(* Logix 5000 project; controller PBS_Perfusion vendor 1 type 14 code 217 rev 32.14; software revision 32.03; part 6 of 27 *)
(* tags used below, declared in another part *)
   Inp_PVSrcQ : DINT;   // Input Source and Quality (from Channel object, if available) (enum)
   Inp_PVNotify : DINT;   // Related PV object alarm prio and ack status (enum)
   Inp_PVBad : BOOL;   // 1=PV or I/O Comms Status Bad, 0=OK
   Inp_PVUncertain : BOOL;   // 1=PV Value Not Reliable, 0=OK
   Inp_Sim : BOOL;   // 1=Use simulated PV (Set_SimPV); 0=Use Input (Inp_PV)
   Cfg_HasRoC : BOOL;   // 1=Enables the Rate of Change calc and HiRoC alarm
   Cfg_HasDev : BOOL;   // 1=Enables Reference entry and Deviation calc and alarms
   Cfg_UseChanSrcQ : BOOL;   // 1=Pass thru connected Channel's SrcQ value, 0=generate SrcQ
   Cfg_RateTime : REAL;   // PV Rate of Change time base (sec) 60=/min, 3600=/hr
   Cfg_Ref : REAL;   // Analog Reference for Deviation Alarms (EU)
   Cfg_CtrlHiHiLim : REAL;   // Current High-High Control Threshold
   Cfg_CtrlHiHiDB : REAL;   // High-High Control Deadband (EU)
   Cfg_CtrlHiLim : REAL;   // Current High Control Threshold
   Cfg_CtrlHiDB : REAL;   // High Control Deadband (EU)
   Cfg_CtrlLoLim : REAL;   // Current Low Control Threshold
   Cfg_CtrlLoDB : REAL;   // Low Control Deadband (EU)
   Cfg_CtrlLoLoLim : REAL;   // Current Low-Low Control Threshold
   Cfg_CtrlLoLoDB : REAL;   // Low-Low Control Deadband (EU)
   Cfg_HiHiLim : REAL;   // Current High-High Status Threshold
   Cfg_HiHiDB : REAL;   // High-High Status Deadband (EU)
   Cfg_HiLim : REAL;   // Current High Status Threshold
   Cfg_HiDB : REAL;   // High Status Deadband (EU)
   Cfg_LoLim : REAL;   // Current Low Status Threshold
   Cfg_LoDB : REAL;   // Low Status Deadband (EU)
   Cfg_LoLoLim : REAL;   // Current Low-Low Status Threshold
   Cfg_LoLoDB : REAL;   // Low-Low Status Deadband (EU)
   Cfg_HiRoCLim : REAL;   // Current High Rate of Change Status Threshold
   Cfg_HiRoCDB : REAL;   // High Rate of Change Status Deadband (EU/rate time)
   Cfg_HiDevLim : REAL;   // Current High Deviation Status Threshold
   Cfg_HiDevDB : REAL;   // High Deviation Status Deadband (EU)
   Cfg_LoDevLim : REAL;   // Current Low Deviation Status Threshold
   Cfg_LoDevDB : REAL;   // Low Deviation Status Deadband (EU)
   Cfg_FailHiLim : REAL;   // Out-of-Range (fail) High Limit (EU)
   Cfg_FailLoLim : REAL;   // Out-of-Range (fail) Low Limit (EU)
   Cfg_FailDB : REAL;   // Out-of-Range (fail) High/Low Deadband (EU)
   PCmd_ClearCapt : BOOL;   // Program Command to Clear the captured min / max PV excursion values
   Val : REAL;   // Analog Input Value (incl. Manual Override, if used)
   Val_InpPV : REAL;   // Analog Input Value (actual, before Substitute PV selection)
   Val_RoC : REAL;   // Analog Value Rate of Change (EU/rate time)
   Val_Dev : REAL;   // Calculated Deviation from Reference (EU)
   Val_PVMinCapt : REAL;   // Captured PV Minimum (excursion) since last cleared
   Val_PVMaxCapt : REAL;   // Captured PV Maximum (excursion) since last cleared
   SrcQ_IO : DINT;   // Source and Quality of primary I/O (enumeration)
   SrcQ : DINT;   // Source and Quality of primary Val/Sts (enumeration)
   Val_Fault : DINT;   // Device Fault Status 0=none, 20=Lo, 21=Hi, 22=LoDev, 23=HiDev, 24=LoLo, 25=HiHi, 26=HiRoC 32=Fail, 34=CfgErr
   Val_NotifyAll : DINT;   // Highest Alarm prio and ack status this object + channel (enum)
   Val_UnackAlmC : DINT;   // Count of Unacknowledged Alarms
   Sts_SubstPV : BOOL;   // 1=Using Substitute PV (Input being overridden)
   Sts_PVBad : BOOL;   // 1=PV Bad quality or Out of Range
   Sts_PVUncertain : BOOL;   // 1=PV Value is Uncertain (quality)
   Sts_AlmInh : BOOL;   // 1=An Alarm is Shelved, Disabled or Suppressed: display icon
   Sts_Err : BOOL;   // 1=Error in Config: see detail bits for reason
   Err_Raw : BOOL;   // 1=Error in Config: Raw Input Scaling Min = Max
   Err_EU : BOOL;   // 1=Error in Config: Scaled EU Min = Max
   Err_Timer : BOOL;   // 1=Error in Config: On-Delay, Off-Delay, Gate Delay Time Invalid (use 0 to 2147483 s)
   Err_Filt : BOOL;   // 1=-Error in Config: PV filter params (RateTime, TC)
   Err_Alarm : BOOL;   // 1=Error in Config: Alarm Min On Time, Shelf Time, Severity
   Sts_RdyReset : ALIAS FOR ORdy_Reset;   // 1=A latched alarm or shed condition is ready to be reset
   Sts_RdyAck : BOOL;   // 1=An alarm is ready to be acknowledged
   Sts_CtrlHiHi : BOOL;   // 1=Analog Input is above High-High Control limit
   Sts_CtrlHi : BOOL;   // 1=Analog Input is above High Control limit
   Sts_CtrlLo : BOOL;   // 1=Analog Input is above Low Control limit
   Sts_CtrlLoLo : BOOL;   // 1=Analog Input is above Low-Low Control limit
   Sts_HiHiCmp : ALIAS FOR HiHiGate.Inp;   // PV High-High comparison result 1=High-High
   Sts_HiHi : ALIAS FOR HiHi.Inp;   // 1=Analog Input is above High-High limit
   Sts_HiCmp : ALIAS FOR HiGate.Inp;   // PV High comparison result 1=High
   Sts_Hi : ALIAS FOR Hi.Inp;   // 1=Analog Input is above High limit
   Sts_LoCmp : ALIAS FOR LoGate.Inp;   // PV Low comparison result 1=Low
   Sts_Lo : ALIAS FOR Lo.Inp;   // 1=Analog Input is below Low limit
   Sts_LoLoCmp : ALIAS FOR LoLoGate.Inp;   // PV Low-Low comparison result 1=Low-Low
   Sts_LoLo : ALIAS FOR LoLo.Inp;   // 1=Analog Input is below Low-Low limit
   Sts_HiRoCCmp : ALIAS FOR HiRoCGate.Inp;   // PV High Rate of Change comparison result 1=High
   Sts_HiRoC : ALIAS FOR HiRoC.Inp;   // 1=Analog Input Rate of Change is above High limit
   Sts_HiDevCmp : ALIAS FOR HiDevGate.Inp;   // PV High Deviation comparison result 1=Dev High
   Sts_HiDev : ALIAS FOR HiDev.Inp;   // 1=Analog Input Deviation is above High limit
   Sts_LoDevCmp : ALIAS FOR LoDevGate.Inp;   // PV Low Deviation comparison result 1=Dev Low
   Sts_LoDev : ALIAS FOR LoDev.Inp;   // 1=Analog Input Deviation is below Low limit
   Sts_FailCmp : ALIAS FOR FailGate.Inp;   // PV Fail comparison result 1=Out of Range
   Sts_Fail : ALIAS FOR Fail.Inp;   // 1=Analog Input is Out of Range or PV Bad
   P_AInAdv : BOOL;   // Unique Parameter Name for auto - discovery
   LoLo : P_Alarm;   // Low-Low Alarm
   Lo : P_Alarm;   // Low Alarm
   Hi : P_Alarm;   // High Alarm
   HiHi : P_Alarm;   // High-High Alarm
   Fail : P_Alarm;   // Analog Input Failure Alarm (bad quality or out of range)
   Wrk_Notify : DINT;   // Buffer for building Val_Notify
   Wrk_Fault : DINT;   // Buffer for building Val_Fault
   Wrk_SrcQ : DINT;   // Register for building Source / Quality enumeration
   Wrk_SubstPV : BOOL;   // Internal flag: Using Substitute PV
   Wrk_ScanTime : REAL;   // Time since this instance was last scanned
   Wrk_RoC : REAL;   // Calculated Rate of Change of PV
   Wrk_PrevPV : REAL;   // Previous scan's value of Filtered PV
   LoDev : P_Alarm;   // Low Deviation Alarm
   HiDev : P_Alarm;   // High Deviation Alarm
   HiRoC : P_Alarm;   // High Rate of Change Alarm
   Wrk_InpInfNaN : BOOL;   // Input (Inp_PV or Set_SimPV) Infinite or Not a Number
   Wrk_SelPVInfNaN : BOOL;   // Selected PV (Input or Substitute) is Infinite or NaN
   Wrk_HiRoC : BOOL;   // Internal flag: High Rate of Change Status
   Wrk_LoDev : BOOL;   // Internal flag: Low Deviation Status
   Wrk_HiDev : BOOL;   // Internal flag: High Deviation Status
   Wrk_Fail : BOOL;   // Internal flag: Fail Status
   Wrk_LoLo : BOOL;   // Internal flag: Low-Low Status
   Wrk_Lo : BOOL;   // Internal flag: Low Status
   Wrk_HiHi : BOOL;   // Internal flag: High-High Status
   Wrk_Hi : BOOL;   // Internal flag: High Status
   LoDevGate : P_Gate;   // Low Deviation Alarm Gate / Delay Block
   HiRoCGate : P_Gate;   // High Rate of Change Alarm Gate / Delay Block
   HiDevGate : P_Gate;   // High Deviation Alarm Gate / Delay Block
   LoLoGate : P_Gate;   // Low-Low Alarm Gate / Delay Block
   LoGate : P_Gate;   // Low Alarm Gate / Delay Block
   HiHiGate : P_Gate;   // High-High Alarm Gate / Delay Block
   HiGate : P_Gate;   // High Alarm Gate / Delay Block
   FailGate : P_Gate;   // Fail Alarm Gate / Delay Block
   Wrk_UnackAlmC : DINT;   // Buffer for building Val_UnackAlmC
   Val_Notify : DINT;   // Highest Alarm prio and ack status this object only (enum)
   OCmd_ClearCapt : BOOL;   // Operator Command to Clear the captured min / max PV excursion values
   ORdy_ResetAckAll : BOOL;   // 1=Ready for OCmd_ResetAckAll (enables HMI button)
   ORdy_Reset : BOOL;   // 1=Ready for OCmd_Reset (enables HMI button)
   Wrk_RawPV : REAL;   // Value of raw PV to be used for Out of Range checking
   REAL : DINT;
(* P_AInAdv, continued *)

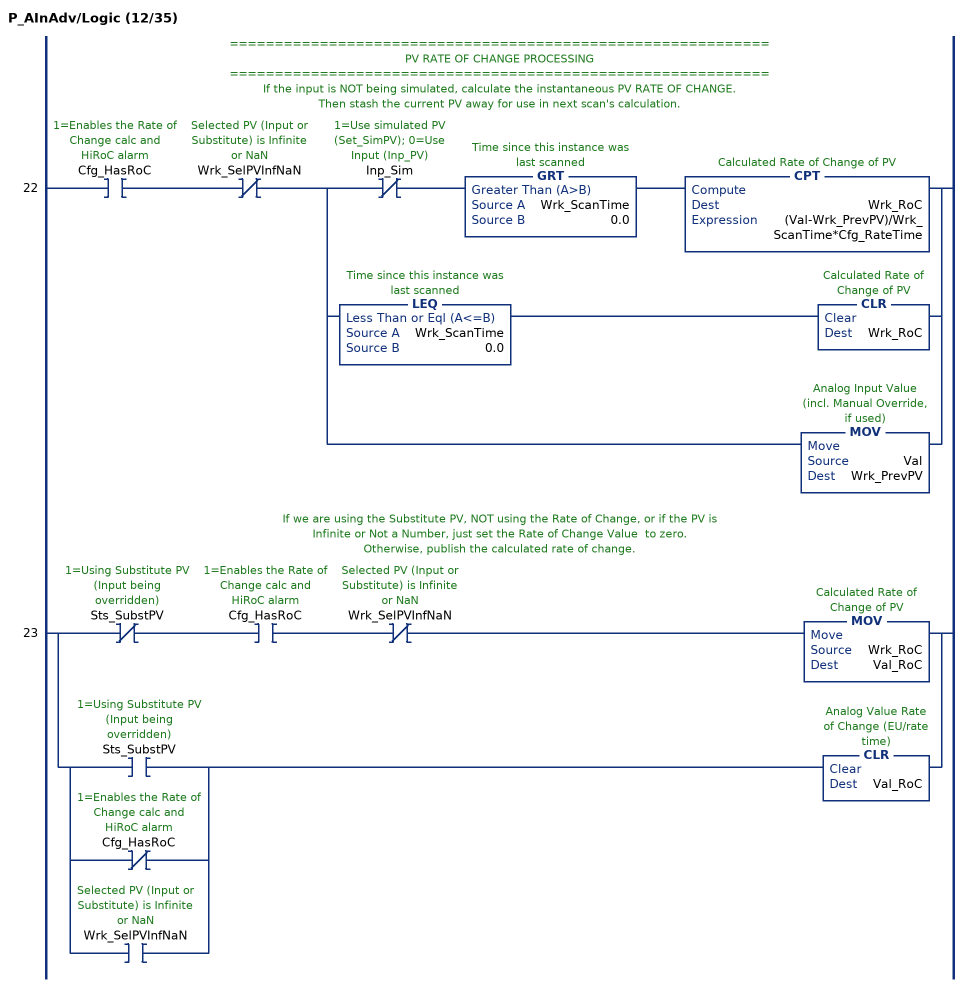
   [picture p107: P_AInAdv/Logic rungs 22-23]
   // ============================================================
   // PV RATE OF CHANGE PROCESSING
   // ============================================================
   // If the input is NOT being simulated, calculate the instantaneous PV RATE OF CHANGE.
   // Then stash the current PV away for use in next scan's calculation.
   22: XIC(Cfg_HasRoC)XIO(Wrk_SelPVInfNaN)[XIO(Inp_Sim) GRT(Wrk_ScanTime,0.0) CPT(Wrk_RoC,(Val-Wrk_PrevPV)/Wrk_ScanTime*Cfg_RateTime) ,LEQ(Wrk_ScanTime,0.0) CLR(Wrk_RoC) ,MOV(Val,Wrk_PrevPV) ];
   // If we are using the Substitute PV, NOT using the Rate of Change, or if the PV is
   // Infinite or Not a Number, just set the Rate of Change Value  to zero.
   // Otherwise, publish the calculated rate of change.
   23: [XIO(Sts_SubstPV) XIC(Cfg_HasRoC) XIO(Wrk_SelPVInfNaN) MOV(Wrk_RoC,Val_RoC) ,[XIC(Sts_SubstPV) ,XIO(Cfg_HasRoC) ,XIC(Wrk_SelPVInfNaN) ] CLR(Val_RoC) ];
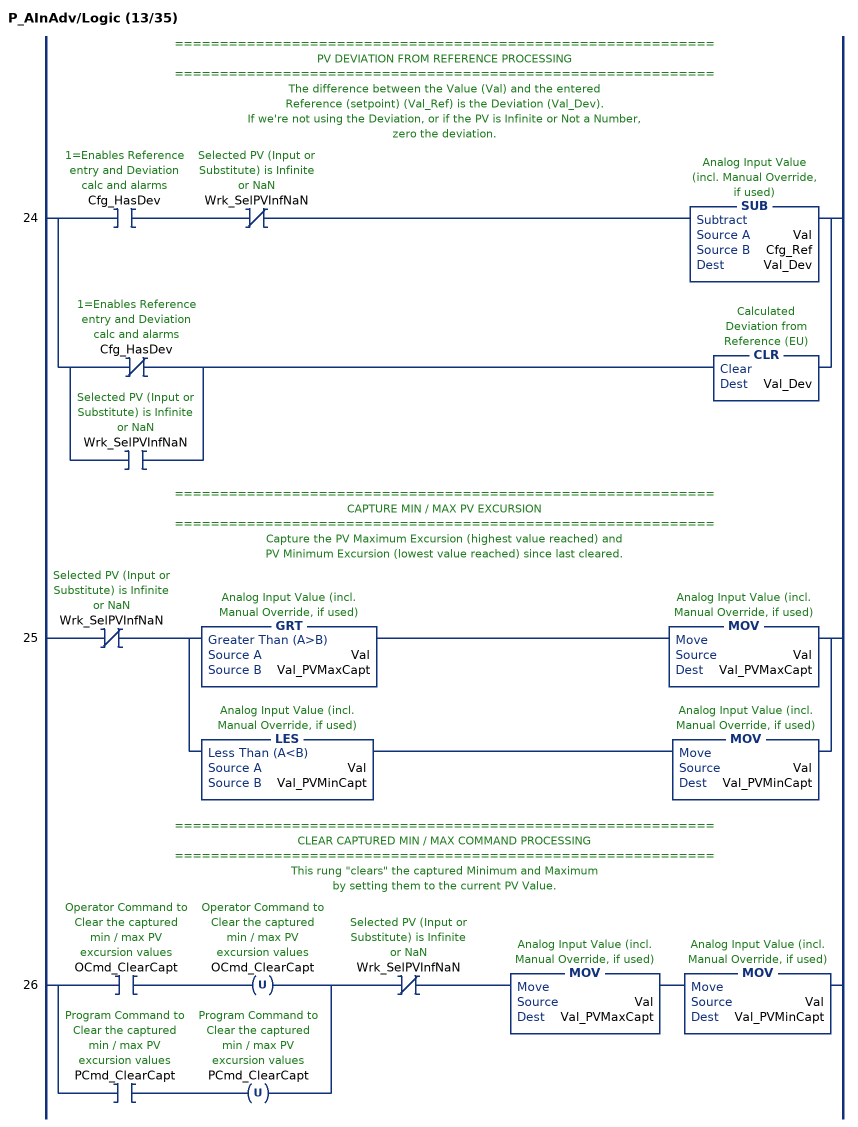
   // ============================================================
   // PV DEVIATION FROM REFERENCE PROCESSING
   // ============================================================
   // The difference between the Value (Val) and the entered
   // Reference (setpoint) (Val_Ref) is the Deviation (Val_Dev).
   // If we're not using the Deviation, or if the PV is Infinite or Not a Number,
   // zero the deviation.
   24: [XIC(Cfg_HasDev) XIO(Wrk_SelPVInfNaN) SUB(Val,Cfg_Ref,Val_Dev) ,[XIO(Cfg_HasDev) ,XIC(Wrk_SelPVInfNaN) ] CLR(Val_Dev) ];
   // ============================================================
   // CAPTURE MIN / MAX PV EXCURSION
   // ============================================================
   // Capture the PV Maximum Excursion (highest value reached) and
   // PV Minimum Excursion (lowest value reached) since last cleared.
   25: XIO(Wrk_SelPVInfNaN)[GRT(Val,Val_PVMaxCapt) MOV(Val,Val_PVMaxCapt) ,LES(Val,Val_PVMinCapt) MOV(Val,Val_PVMinCapt) ];
   // ============================================================
   // CLEAR CAPTURED MIN / MAX COMMAND PROCESSING
   // ============================================================
   // This rung "clears" the captured Minimum and Maximum
   // by setting them to the current PV Value.
   26: [XIC(OCmd_ClearCapt) OTU(OCmd_ClearCapt) ,XIC(PCmd_ClearCapt) OTU(PCmd_ClearCapt) ]XIO(Wrk_SelPVInfNaN)MOV(Val,Val_PVMaxCapt)MOV(Val,Val_PVMinCapt);
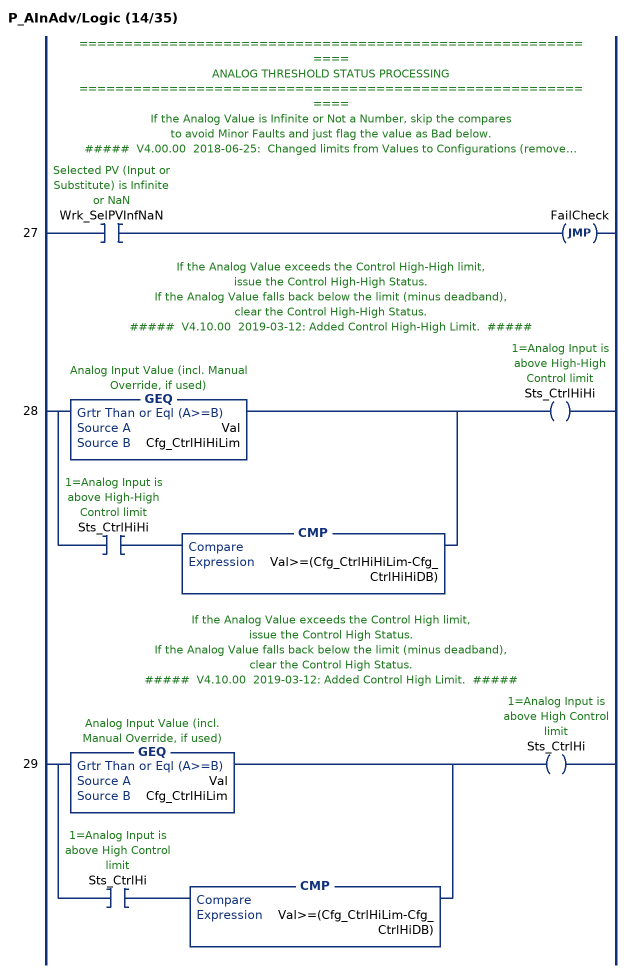
   // ============================================================
   // ANALOG THRESHOLD STATUS PROCESSING
   // ============================================================
   // If the Analog Value is Infinite or Not a Number, skip the compares
   // to avoid Minor Faults and just flag the value as Bad below.
   // #####  V4.00.00  2018-06-25:  Changed limits from Values to Configurations (removed Mode, Settings).  #####
   // #####  Changed PV Out of Range comparisons to use RAW (INPUT) PV, not scaled/filtered value (Val).  #####
   27: XIC(Wrk_SelPVInfNaN)JMP(FailCheck);
   // If the Analog Value exceeds the Control High-High limit,
   // issue the Control High-High Status.
   // If the Analog Value falls back below the limit (minus deadband),
   // clear the Control High-High Status.
   // #####  V4.10.00  2019-03-12: Added Control High-High Limit.  #####
   28: [GEQ(Val,Cfg_CtrlHiHiLim) ,XIC(Sts_CtrlHiHi) CMP(Val>=(Cfg_CtrlHiHiLim-Cfg_CtrlHiHiDB)) ]OTE(Sts_CtrlHiHi);
   // If the Analog Value exceeds the Control High limit,
   // issue the Control High Status.
   // If the Analog Value falls back below the limit (minus deadband),
   // clear the Control High Status.
   // #####  V4.10.00  2019-03-12: Added Control High Limit.  #####
   29: [GEQ(Val,Cfg_CtrlHiLim) ,XIC(Sts_CtrlHi) CMP(Val>=(Cfg_CtrlHiLim-Cfg_CtrlHiDB)) ]OTE(Sts_CtrlHi);
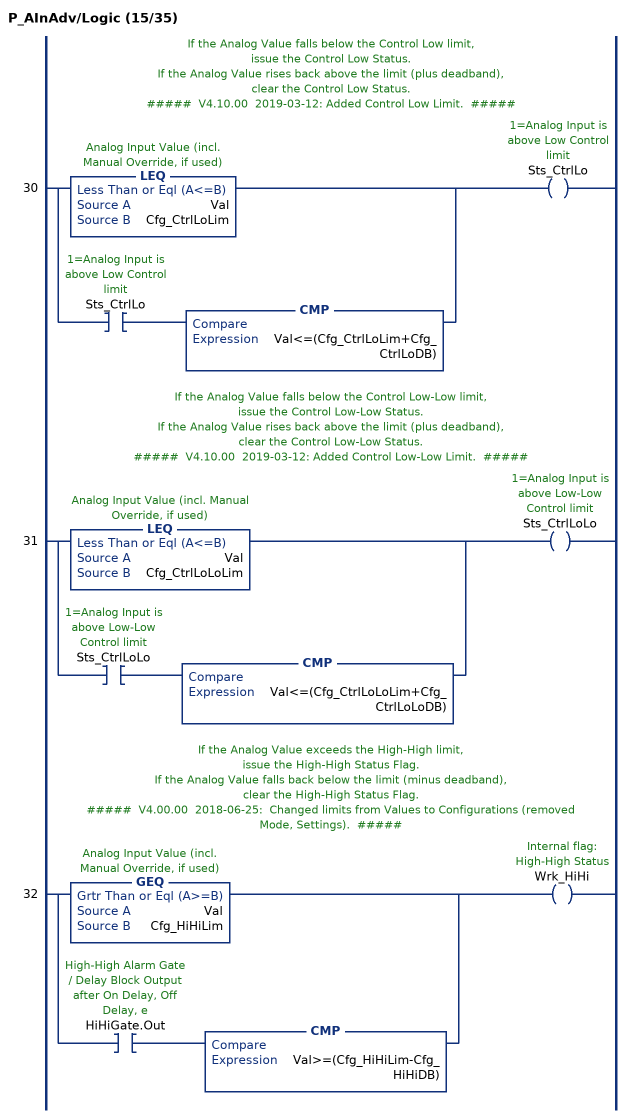
   // If the Analog Value falls below the Control Low limit,
   // issue the Control Low Status.
   // If the Analog Value rises back above the limit (plus deadband),
   // clear the Control Low Status.
   // #####  V4.10.00  2019-03-12: Added Control Low Limit.  #####
   30: [LEQ(Val,Cfg_CtrlLoLim) ,XIC(Sts_CtrlLo) CMP(Val<=(Cfg_CtrlLoLim+Cfg_CtrlLoDB)) ]OTE(Sts_CtrlLo);
   // If the Analog Value falls below the Control Low-Low limit,
   // issue the Control Low-Low Status.
   // If the Analog Value rises back above the limit (plus deadband),
   // clear the Control Low-Low Status.
   // #####  V4.10.00  2019-03-12: Added Control Low-Low Limit.  #####
   31: [LEQ(Val,Cfg_CtrlLoLoLim) ,XIC(Sts_CtrlLoLo) CMP(Val<=(Cfg_CtrlLoLoLim+Cfg_CtrlLoLoDB)) ]OTE(Sts_CtrlLoLo);
   // If the Analog Value exceeds the High-High limit,
   // issue the High-High Status Flag.
   // If the Analog Value falls back below the limit (minus deadband),
   // clear the High-High Status Flag.
   // #####  V4.00.00  2018-06-25:  Changed limits from Values to Configurations (removed Mode, Settings).  #####
   32: [GEQ(Val,Cfg_HiHiLim) ,XIC(HiHiGate.Out) CMP(Val>=(Cfg_HiHiLim-Cfg_HiHiDB)) ]OTE(Wrk_HiHi);
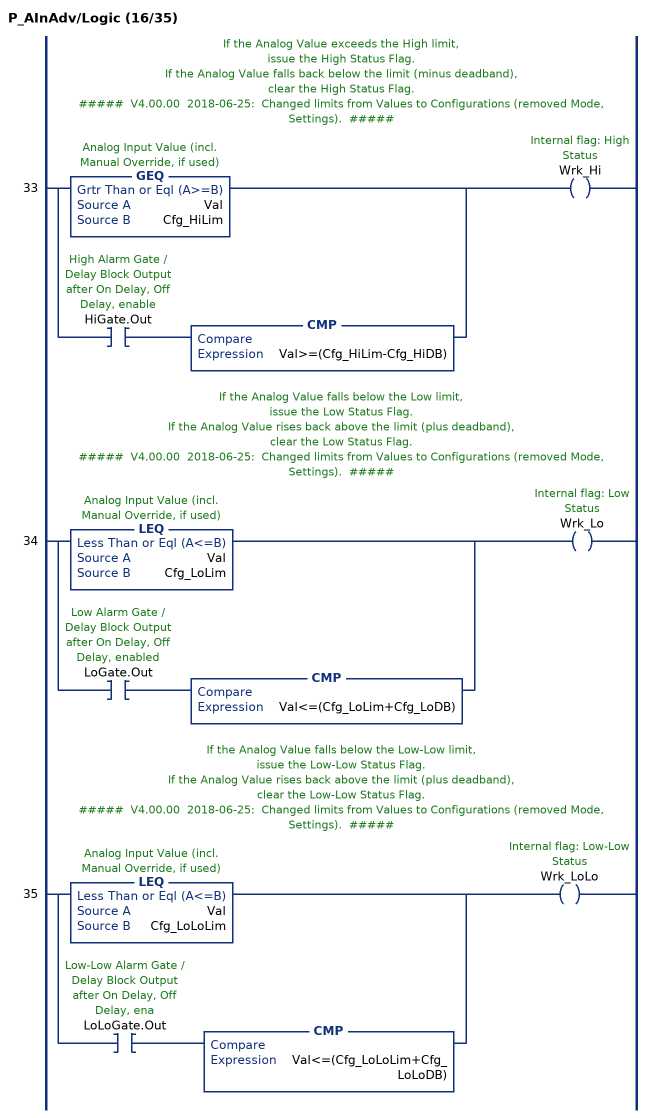
   // If the Analog Value exceeds the High limit,
   // issue the High Status Flag.
   // If the Analog Value falls back below the limit (minus deadband),
   // clear the High Status Flag.
   // #####  V4.00.00  2018-06-25:  Changed limits from Values to Configurations (removed Mode, Settings).  #####
   33: [GEQ(Val,Cfg_HiLim) ,XIC(HiGate.Out) CMP(Val>=(Cfg_HiLim-Cfg_HiDB)) ]OTE(Wrk_Hi);
   // If the Analog Value falls below the Low limit,
   // issue the Low Status Flag.
   // If the Analog Value rises back above the limit (plus deadband),
   // clear the Low Status Flag.
   // #####  V4.00.00  2018-06-25:  Changed limits from Values to Configurations (removed Mode, Settings).  #####
   34: [LEQ(Val,Cfg_LoLim) ,XIC(LoGate.Out) CMP(Val<=(Cfg_LoLim+Cfg_LoDB)) ]OTE(Wrk_Lo);
   // If the Analog Value falls below the Low-Low limit,
   // issue the Low-Low Status Flag.
   // If the Analog Value rises back above the limit (plus deadband),
   // clear the Low-Low Status Flag.
   // #####  V4.00.00  2018-06-25:  Changed limits from Values to Configurations (removed Mode, Settings).  #####
   35: [LEQ(Val,Cfg_LoLoLim) ,XIC(LoLoGate.Out) CMP(Val<=(Cfg_LoLoLim+Cfg_LoLoDB)) ]OTE(Wrk_LoLo);
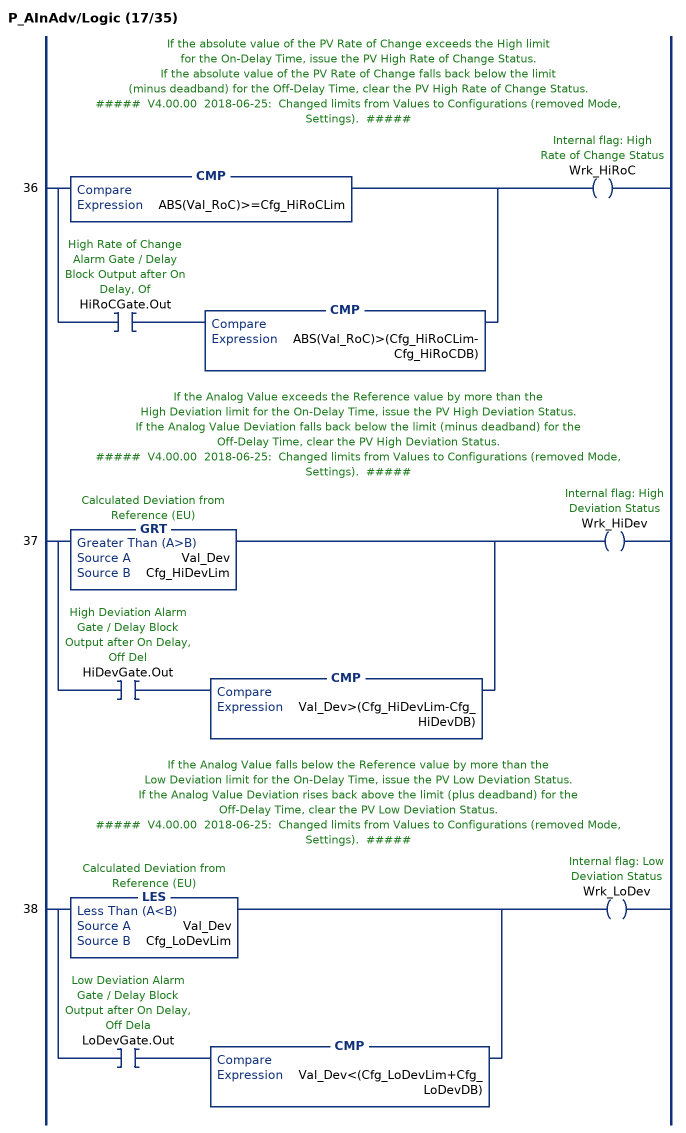
   // If the absolute value of the PV Rate of Change exceeds the High limit
   // for the On-Delay Time, issue the PV High Rate of Change Status.
   // If the absolute value of the PV Rate of Change falls back below the limit
   // (minus deadband) for the Off-Delay Time, clear the PV High Rate of Change Status.
   // #####  V4.00.00  2018-06-25:  Changed limits from Values to Configurations (removed Mode, Settings).  #####
   36: [CMP(ABS(Val_RoC)>=Cfg_HiRoCLim) ,XIC(HiRoCGate.Out) CMP(ABS(Val_RoC)>(Cfg_HiRoCLim-Cfg_HiRoCDB)) ]OTE(Wrk_HiRoC);
   // If the Analog Value exceeds the Reference value by more than the
   // High Deviation limit for the On-Delay Time, issue the PV High Deviation Status.
   // If the Analog Value Deviation falls back below the limit (minus deadband) for the
   // Off-Delay Time, clear the PV High Deviation Status.
   // #####  V4.00.00  2018-06-25:  Changed limits from Values to Configurations (removed Mode, Settings).  #####
   37: [GRT(Val_Dev,Cfg_HiDevLim) ,XIC(HiDevGate.Out) CMP(Val_Dev>(Cfg_HiDevLim-Cfg_HiDevDB)) ]OTE(Wrk_HiDev);
   // If the Analog Value falls below the Reference value by more than the
   // Low Deviation limit for the On-Delay Time, issue the PV Low Deviation Status.
   // If the Analog Value Deviation rises back above the limit (plus deadband) for the
   // Off-Delay Time, clear the PV Low Deviation Status.
   // #####  V4.00.00  2018-06-25:  Changed limits from Values to Configurations (removed Mode, Settings).  #####
   38: [LES(Val_Dev,Cfg_LoDevLim) ,XIC(LoDevGate.Out) CMP(Val_Dev<(Cfg_LoDevLim+Cfg_LoDevDB)) ]OTE(Wrk_LoDev);
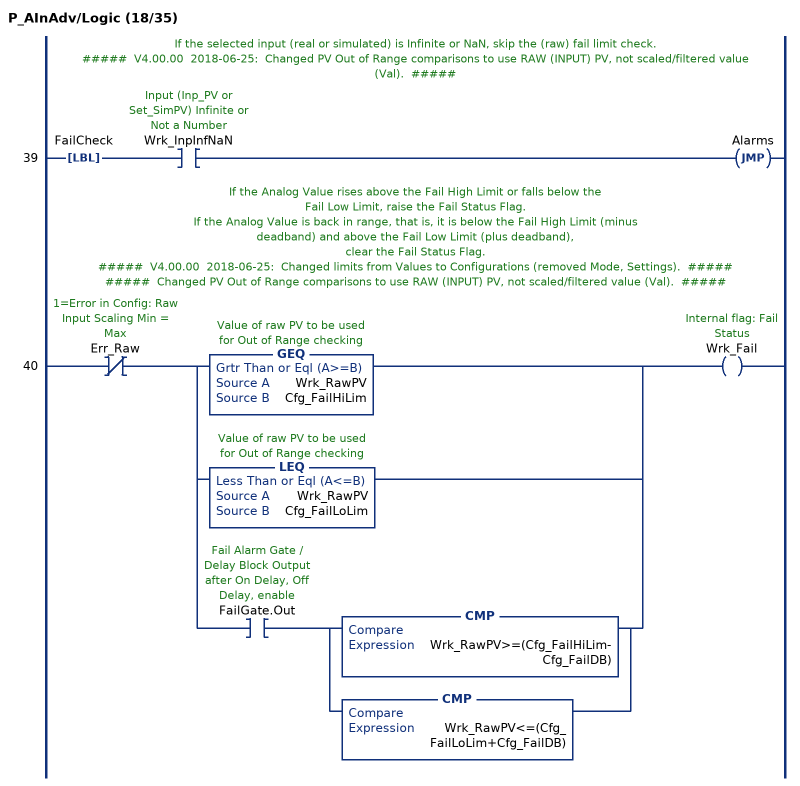
   // If the selected input (real or simulated) is Infinite or NaN, skip the (raw) fail limit check.
   // #####  V4.00.00  2018-06-25:  Changed PV Out of Range comparisons to use RAW (INPUT) PV, not scaled/filtered value (Val).  #####
   39: LBL(FailCheck)XIC(Wrk_InpInfNaN)JMP(Alarms);
   // If the Analog Value rises above the Fail High Limit or falls below the
   // Fail Low Limit, raise the Fail Status Flag.
   // If the Analog Value is back in range, that is, it is below the Fail High Limit (minus
   // deadband) and above the Fail Low Limit (plus deadband),
   // clear the Fail Status Flag.
   // #####  V4.00.00  2018-06-25:  Changed limits from Values to Configurations (removed Mode, Settings).  #####
   // #####  Changed PV Out of Range comparisons to use RAW (INPUT) PV, not scaled/filtered value (Val).  #####
   40: XIO(Err_Raw)[[GEQ(Wrk_RawPV,Cfg_FailHiLim) ,LEQ(Wrk_RawPV,Cfg_FailLoLim) ] ,XIC(FailGate.Out) [CMP(Wrk_RawPV>=(Cfg_FailHiLim-Cfg_FailDB)) ,CMP(Wrk_RawPV<=(Cfg_FailLoLim+Cfg_FailDB)) ] ]OTE(Wrk_Fail);
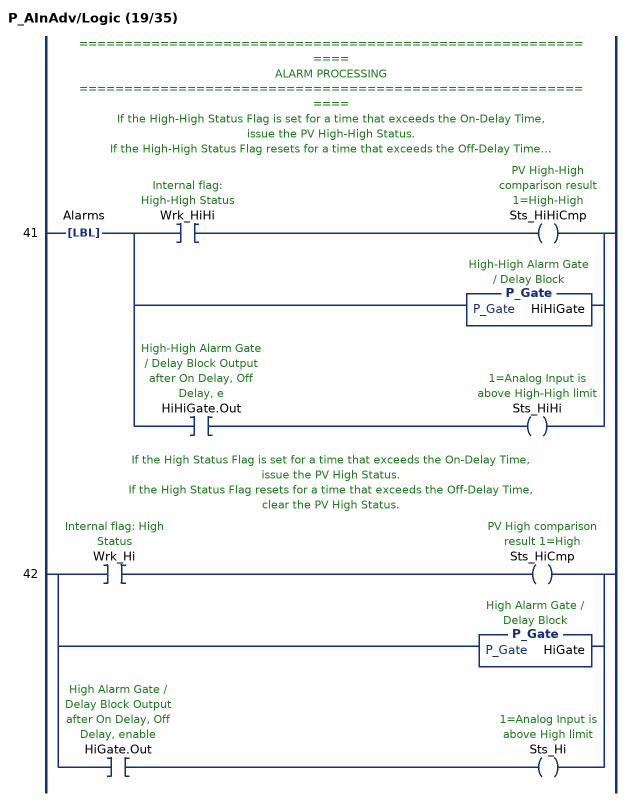
   // ============================================================
   // ALARM PROCESSING
   // ============================================================
   // If the High-High Status Flag is set for a time that exceeds the On-Delay Time,
   // issue the PV High-High Status.
   // If the High-High Status Flag resets for a time that exceeds the Off-Delay Time,
   // clear the PV High-High Status.
   41: LBL(Alarms)[XIC(Wrk_HiHi) OTE(Sts_HiHiCmp) ,P_Gate(HiHiGate) ,XIC(HiHiGate.Out) OTE(Sts_HiHi) ];
   // If the High Status Flag is set for a time that exceeds the On-Delay Time,
   // issue the PV High Status.
   // If the High Status Flag resets for a time that exceeds the Off-Delay Time,
   // clear the PV High Status.
   42: [XIC(Wrk_Hi) OTE(Sts_HiCmp) ,P_Gate(HiGate) ,XIC(HiGate.Out) OTE(Sts_Hi) ];
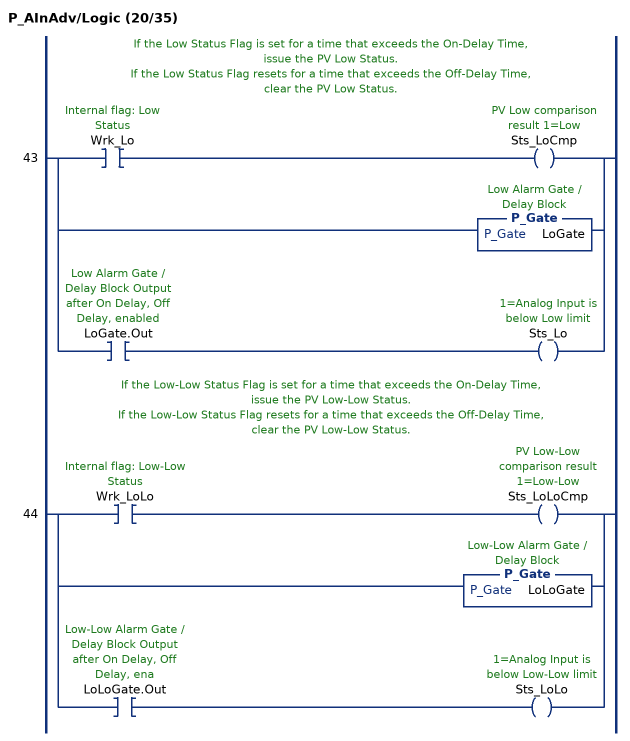
   // If the Low Status Flag is set for a time that exceeds the On-Delay Time,
   // issue the PV Low Status.
   // If the Low Status Flag resets for a time that exceeds the Off-Delay Time,
   // clear the PV Low Status.
   43: [XIC(Wrk_Lo) OTE(Sts_LoCmp) ,P_Gate(LoGate) ,XIC(LoGate.Out) OTE(Sts_Lo) ];
   // If the Low-Low Status Flag is set for a time that exceeds the On-Delay Time,
   // issue the PV Low-Low Status.
   // If the Low-Low Status Flag resets for a time that exceeds the Off-Delay Time,
   // clear the PV Low-Low Status.
   44: [XIC(Wrk_LoLo) OTE(Sts_LoLoCmp) ,P_Gate(LoLoGate) ,XIC(LoLoGate.Out) OTE(Sts_LoLo) ];
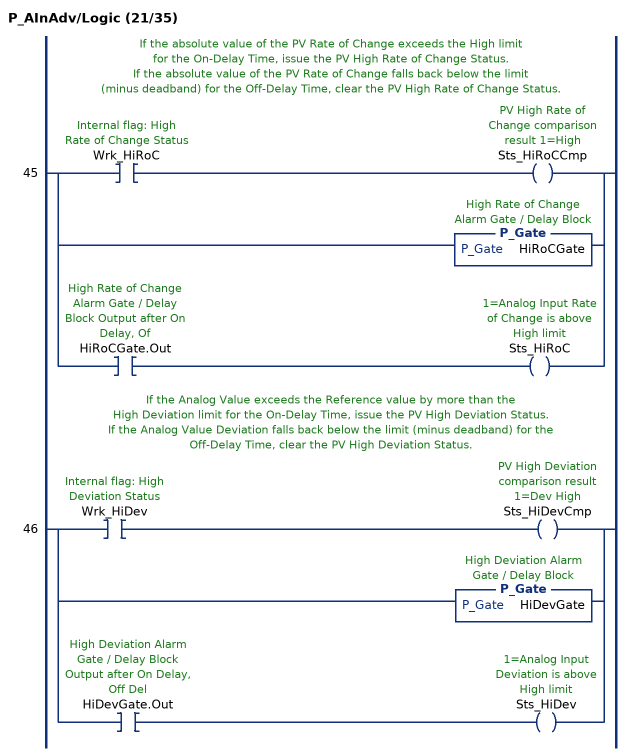
   // If the absolute value of the PV Rate of Change exceeds the High limit
   // for the On-Delay Time, issue the PV High Rate of Change Status.
   // If the absolute value of the PV Rate of Change falls back below the limit
   // (minus deadband) for the Off-Delay Time, clear the PV High Rate of Change Status.
   45: [XIC(Wrk_HiRoC) OTE(Sts_HiRoCCmp) ,P_Gate(HiRoCGate) ,XIC(HiRoCGate.Out) OTE(Sts_HiRoC) ];
   // If the Analog Value exceeds the Reference value by more than the
   // High Deviation limit for the On-Delay Time, issue the PV High Deviation Status.
   // If the Analog Value Deviation falls back below the limit (minus deadband) for the
   // Off-Delay Time, clear the PV High Deviation Status.
   46: [XIC(Wrk_HiDev) OTE(Sts_HiDevCmp) ,P_Gate(HiDevGate) ,XIC(HiDevGate.Out) OTE(Sts_HiDev) ];
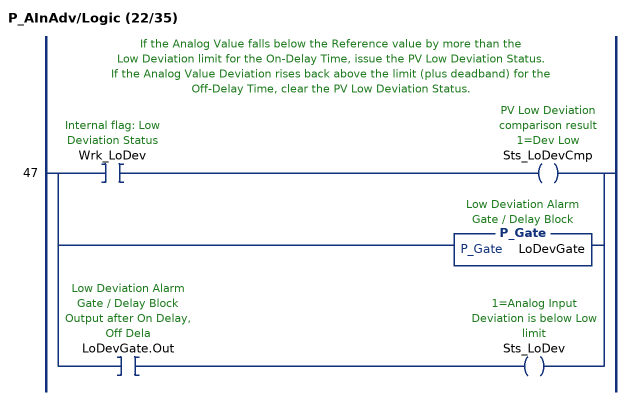
   // If the Analog Value falls below the Reference value by more than the
   // Low Deviation limit for the On-Delay Time, issue the PV Low Deviation Status.
   // If the Analog Value Deviation rises back above the limit (plus deadband) for the
   // Off-Delay Time, clear the PV Low Deviation Status.
   47: [XIC(Wrk_LoDev) OTE(Sts_LoDevCmp) ,P_Gate(LoDevGate) ,XIC(LoDevGate.Out) OTE(Sts_LoDev) ];
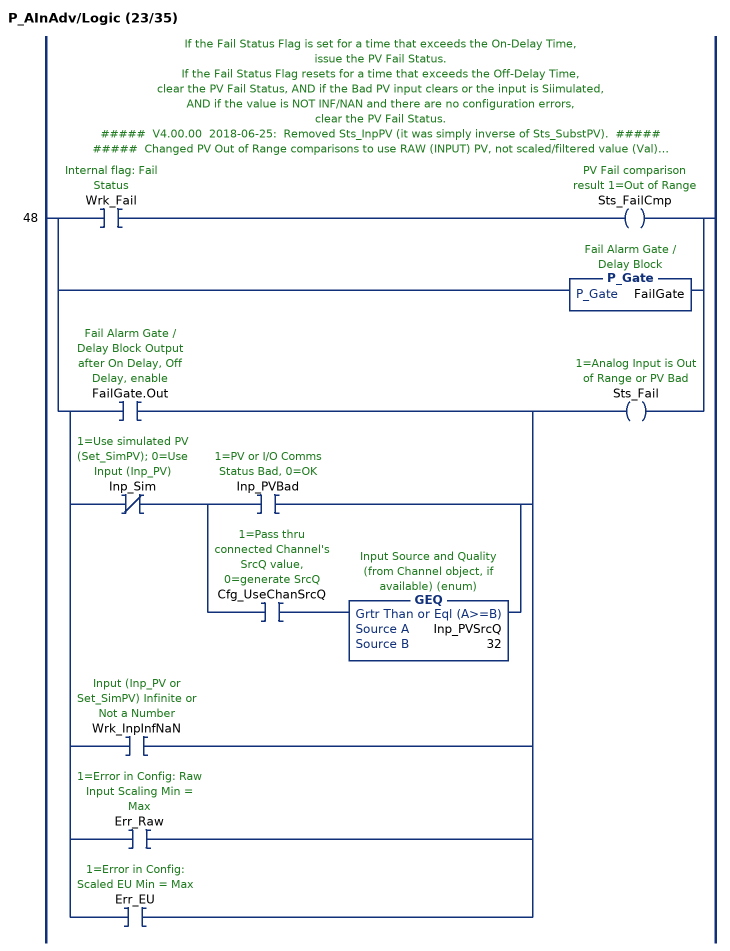
   // If the Fail Status Flag is set for a time that exceeds the On-Delay Time,
   // issue the PV Fail Status.
   // If the Fail Status Flag resets for a time that exceeds the Off-Delay Time,
   // clear the PV Fail Status, AND if the Bad PV input clears or the input is Siimulated,
   // AND if the value is NOT INF/NAN and there are no configuration errors,
   // clear the PV Fail Status.
   // #####  V4.00.00  2018-06-25:  Removed Sts_InpPV (it was simply inverse of Sts_SubstPV).  #####
   // #####  Changed PV Out of Range comparisons to use RAW (INPUT) PV, not scaled/filtered value (Val).  #####
   48: [XIC(Wrk_Fail) OTE(Sts_FailCmp) ,P_Gate(FailGate) ,[XIC(FailGate.Out) ,XIO(Inp_Sim) [XIC(Inp_PVBad) ,XIC(Cfg_UseChanSrcQ) GEQ(Inp_PVSrcQ,32) ] ,XIC(Wrk_InpInfNaN) ,XIC(Err_Raw) ,XIC(Err_EU) ] OTE(Sts_Fail) ];
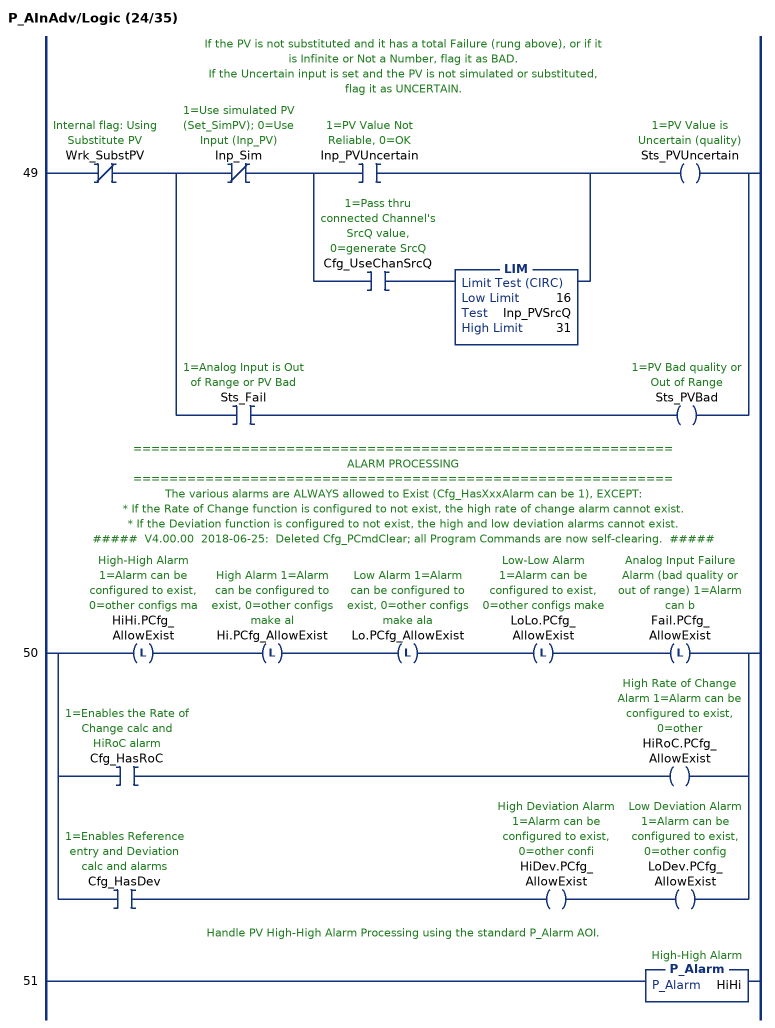
   // If the PV is not substituted and it has a total Failure (rung above), or if it
   // is Infinite or Not a Number, flag it as BAD.
   // If the Uncertain input is set and the PV is not simulated or substituted,
   // flag it as UNCERTAIN.
   49: XIO(Wrk_SubstPV)[XIO(Inp_Sim) [XIC(Inp_PVUncertain) ,XIC(Cfg_UseChanSrcQ) LIM(16,Inp_PVSrcQ,31) ] OTE(Sts_PVUncertain) ,XIC(Sts_Fail) OTE(Sts_PVBad) ];
   // ============================================================
   // ALARM PROCESSING
   // ============================================================
   // The various alarms are ALWAYS allowed to Exist (Cfg_HasXxxAlarm can be 1), EXCEPT:
   // * If the Rate of Change function is configured to not exist, the high rate of change alarm cannot exist.
   // * If the Deviation function is configured to not exist, the high and low deviation alarms cannot exist.
   // #####  V4.00.00  2018-06-25:  Deleted Cfg_PCmdClear; all Program Commands are now self-clearing.  #####
   50: [OTL(HiHi.PCfg_AllowExist) OTL(Hi.PCfg_AllowExist) OTL(Lo.PCfg_AllowExist) OTL(LoLo.PCfg_AllowExist) OTL(Fail.PCfg_AllowExist) ,XIC(Cfg_HasRoC) OTE(HiRoC.PCfg_AllowExist) ,XIC(Cfg_HasDev) OTE(HiDev.PCfg_AllowExist) OTE(LoDev.PCfg_AllowExist) ];
   // Handle PV High-High Alarm Processing using the standard P_Alarm AOI.
   51: P_Alarm(HiHi);
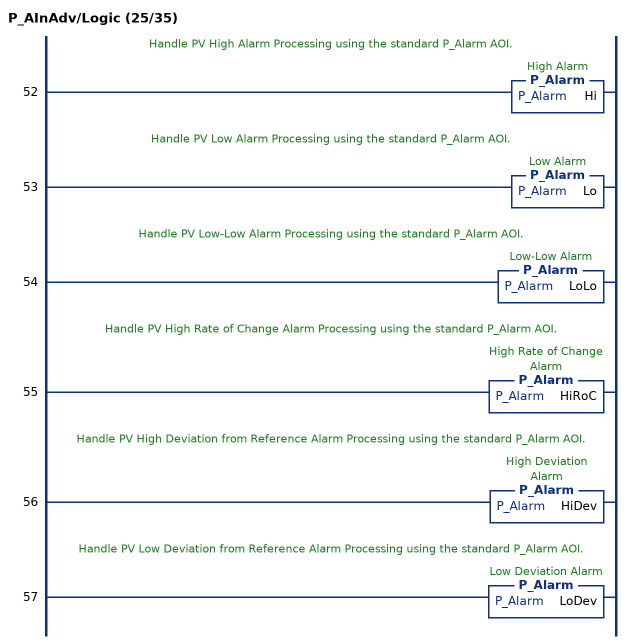
   // Handle PV High Alarm Processing using the standard P_Alarm AOI.
   52: P_Alarm(Hi);
   // Handle PV Low Alarm Processing using the standard P_Alarm AOI.
   53: P_Alarm(Lo);
   // Handle PV Low-Low Alarm Processing using the standard P_Alarm AOI.
   54: P_Alarm(LoLo);
   // Handle PV High Rate of Change Alarm Processing using the standard P_Alarm AOI.
   55: P_Alarm(HiRoC);
   // Handle PV High Deviation from Reference Alarm Processing using the standard P_Alarm AOI.
   56: P_Alarm(HiDev);
   // Handle PV Low Deviation from Reference Alarm Processing using the standard P_Alarm AOI.
   57: P_Alarm(LoDev);
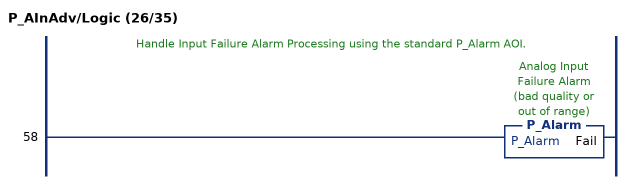
   // Handle Input Failure Alarm Processing using the standard P_Alarm AOI.
   58: P_Alarm(Fail);
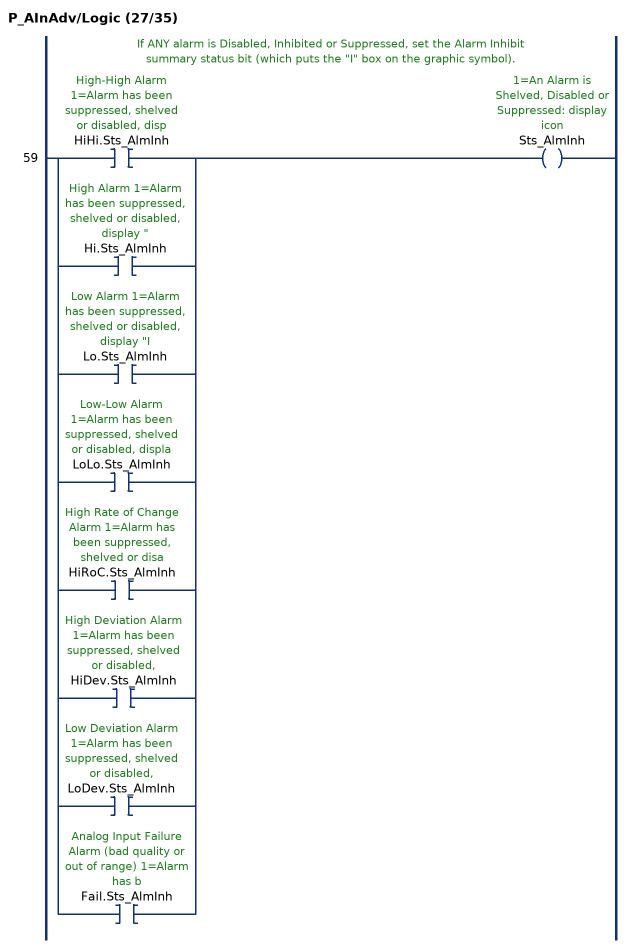
   // If ANY alarm is Disabled, Inhibited or Suppressed, set the Alarm Inhibit
   // summary status bit (which puts the "I" box on the graphic symbol).
   59: [XIC(HiHi.Sts_AlmInh) ,XIC(Hi.Sts_AlmInh) ,XIC(Lo.Sts_AlmInh) ,XIC(LoLo.Sts_AlmInh) ,XIC(HiRoC.Sts_AlmInh) ,XIC(HiDev.Sts_AlmInh) ,XIC(LoDev.Sts_AlmInh) ,XIC(Fail.Sts_AlmInh) ]OTE(Sts_AlmInh);
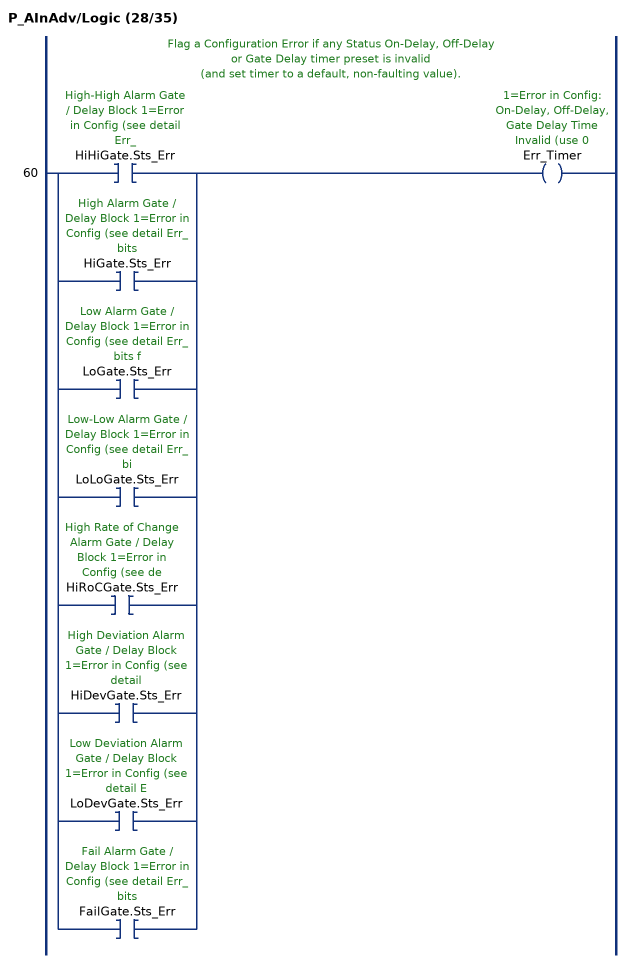
   // Flag a Configuration Error if any Status On-Delay, Off-Delay
   // or Gate Delay timer preset is invalid
   // (and set timer to a default, non-faulting value).
   60: [XIC(HiHiGate.Sts_Err) ,XIC(HiGate.Sts_Err) ,XIC(LoGate.Sts_Err) ,XIC(LoLoGate.Sts_Err) ,XIC(HiRoCGate.Sts_Err) ,XIC(HiDevGate.Sts_Err) ,XIC(LoDevGate.Sts_Err) ,XIC(FailGate.Sts_Err) ]OTE(Err_Timer);
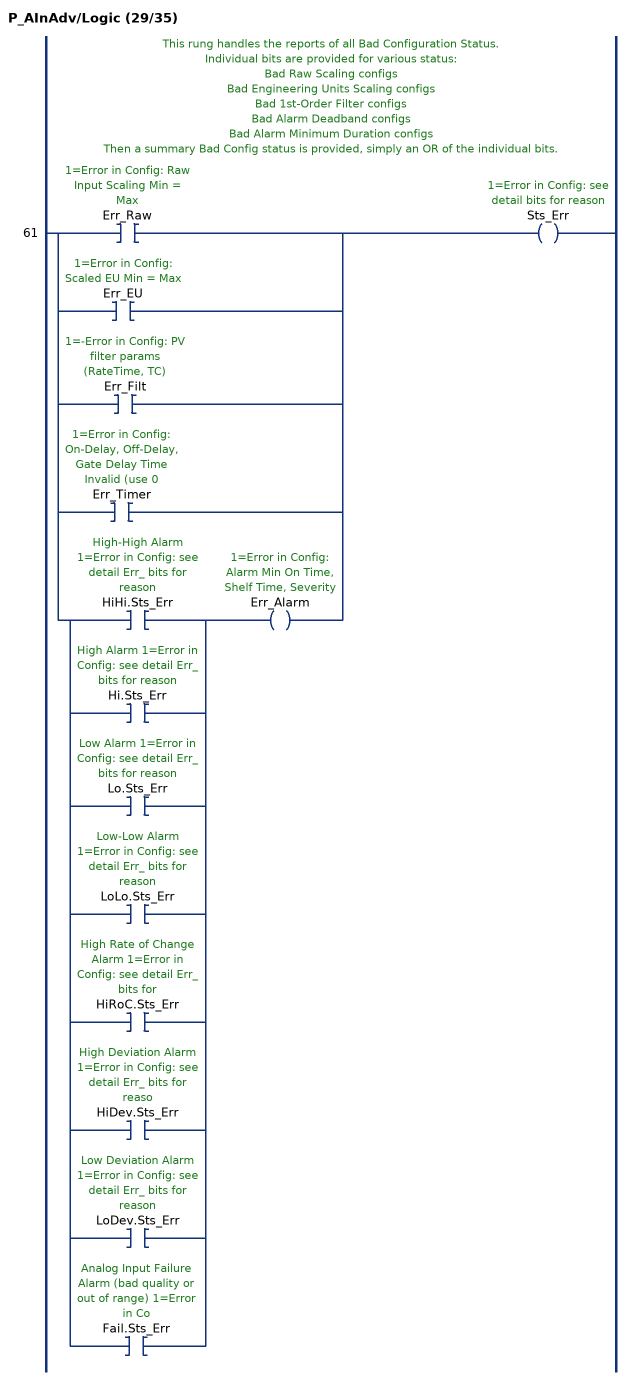
   // This rung handles the reports of all Bad Configuration Status.
   // Individual bits are provided for various status:
   // Bad Raw Scaling configs
   // Bad Engineering Units Scaling configs
   // Bad 1st-Order Filter configs
   // Bad Alarm Deadband configs
   // Bad Alarm Minimum Duration configs
   // Then a summary Bad Config status is provided, simply an OR of the individual bits.
   61: [XIC(Err_Raw) ,XIC(Err_EU) ,XIC(Err_Filt) ,XIC(Err_Timer) ,[XIC(HiHi.Sts_Err) ,XIC(Hi.Sts_Err) ,XIC(Lo.Sts_Err) ,XIC(LoLo.Sts_Err) ,XIC(HiRoC.Sts_Err) ,XIC(HiDev.Sts_Err) ,XIC(LoDev.Sts_Err) ,XIC(Fail.Sts_Err) ] OTE(Err_Alarm) ]OTE(Sts_Err);
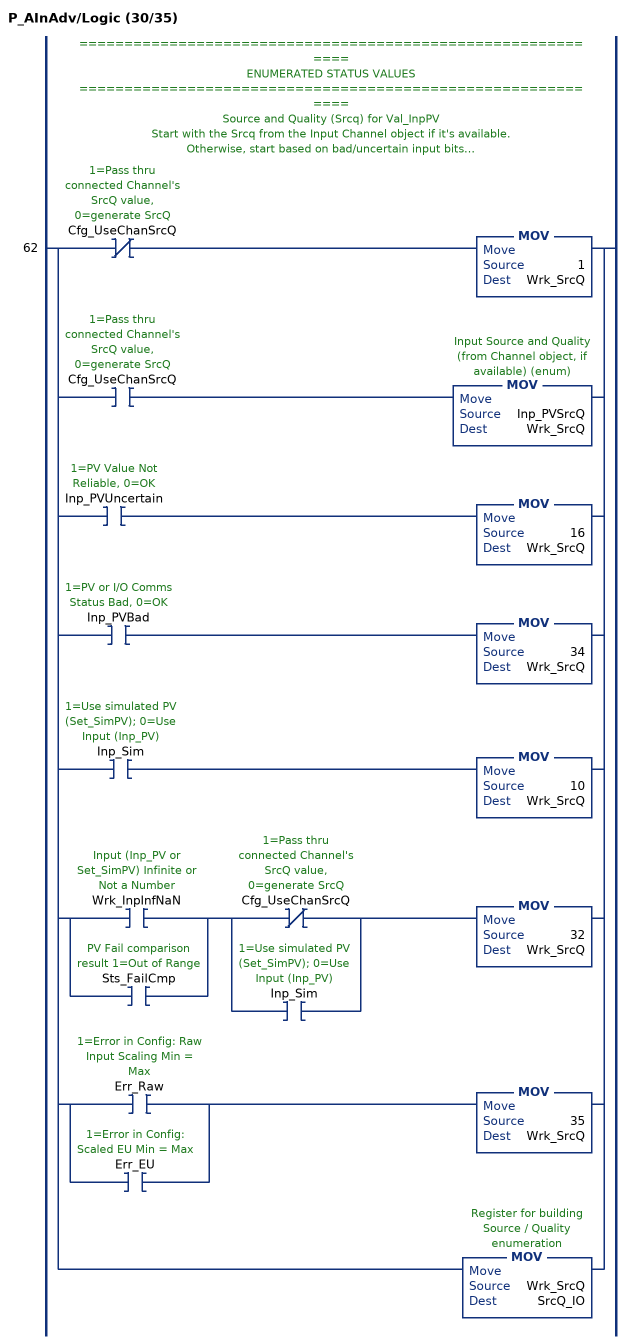
   // ============================================================
   // ENUMERATED STATUS VALUES
   // ============================================================
   // Source and Quality (Srcq) for Val_InpPV
   // Start with the Srcq from the Input Channel object if it's available.
   // Otherwise, start based on bad/uncertain input bits.
   // 0 = Good: live, confirmed good;   1 = Good: live, assumed good;
   // 2 = Good: no feedback, assumed good;   8 = Test: Simulated;   9 = Test: Loopback;
   // 10 = Test: Manually Entered;   16 = Uncertain: Live, off-spec;
   // 17 = Uncertain, Substituted at Device / Bus;   18 = Uncertain, Substituted at AOI;
   // 19 = Uncertain, using last known good;    20 = Uncertain, using replacement value;
   // 32 = Bad, Signal Failure;   33 = Bad, Channel Fault;
   // 34 = Bad, Module / Comms Fault;   35 = Bad, Invalid Configuration
   // #####  V4.00.00  2018-06-25:  Modified to correct precedence and value of Simulated PV.  #####
   // #####  V4.00.01  2018-08-29:  Modified handling of Simulated PV and scaling config errors.  #####
   62: [XIO(Cfg_UseChanSrcQ) MOV(1,Wrk_SrcQ) ,XIC(Cfg_UseChanSrcQ) MOV(Inp_PVSrcQ,Wrk_SrcQ) ,XIC(Inp_PVUncertain) MOV(16,Wrk_SrcQ) ,XIC(Inp_PVBad) MOV(34,Wrk_SrcQ) ,XIC(Inp_Sim) MOV(10,Wrk_SrcQ) ,[XIC(Wrk_InpInfNaN) ,XIC(Sts_FailCmp) ] [XIO(Cfg_UseChanSrcQ) ,XIC(Inp_Sim) ] MOV(32,Wrk_SrcQ) ,[XIC(Err_Raw) ,XIC(Err_EU) ] MOV(35,Wrk_SrcQ) ,MOV(Wrk_SrcQ,SrcQ_IO) ];
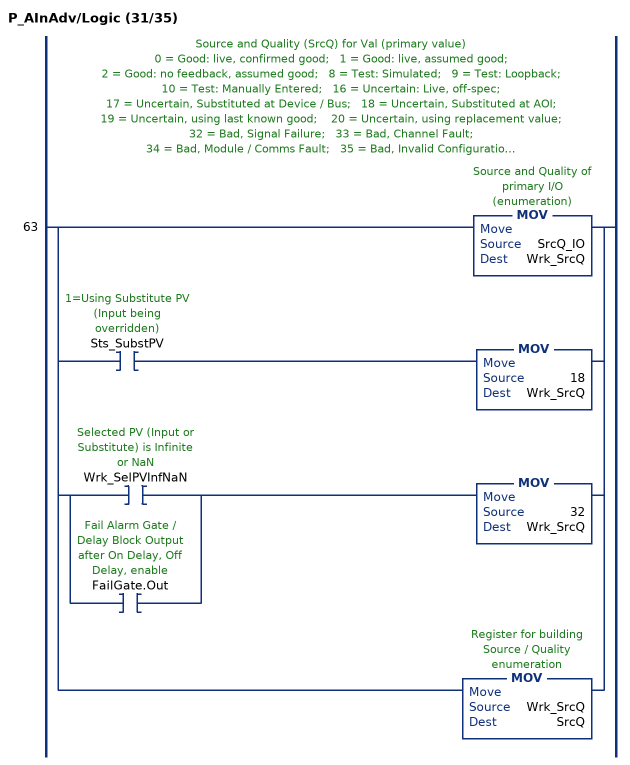
   // Source and Quality (SrcQ) for Val (primary value)
   // 0 = Good: live, confirmed good;   1 = Good: live, assumed good;
   // 2 = Good: no feedback, assumed good;   8 = Test: Simulated;   9 = Test: Loopback;
   // 10 = Test: Manually Entered;   16 = Uncertain: Live, off-spec;
   // 17 = Uncertain, Substituted at Device / Bus;   18 = Uncertain, Substituted at AOI;
   // 19 = Uncertain, using last known good;    20 = Uncertain, using replacement value;
   // 32 = Bad, Signal Failure;   33 = Bad, Channel Fault;
   // 34 = Bad, Module / Comms Fault;   35 = Bad, Invalid Configuration
   // #####  V4.00.00  2018-06-25:  Modified to allow Substitute PV to control SrcQ despite alarm for failed PV.  #####
   // #####  V4.00.01  2018-08-29:  Modified handling of Substitute PV and Channel SrcQ.  #####
   63: [MOV(SrcQ_IO,Wrk_SrcQ) ,XIC(Sts_SubstPV) MOV(18,Wrk_SrcQ) ,[XIC(Wrk_SelPVInfNaN) ,XIC(FailGate.Out) ] MOV(32,Wrk_SrcQ) ,MOV(Wrk_SrcQ,SrcQ) ];
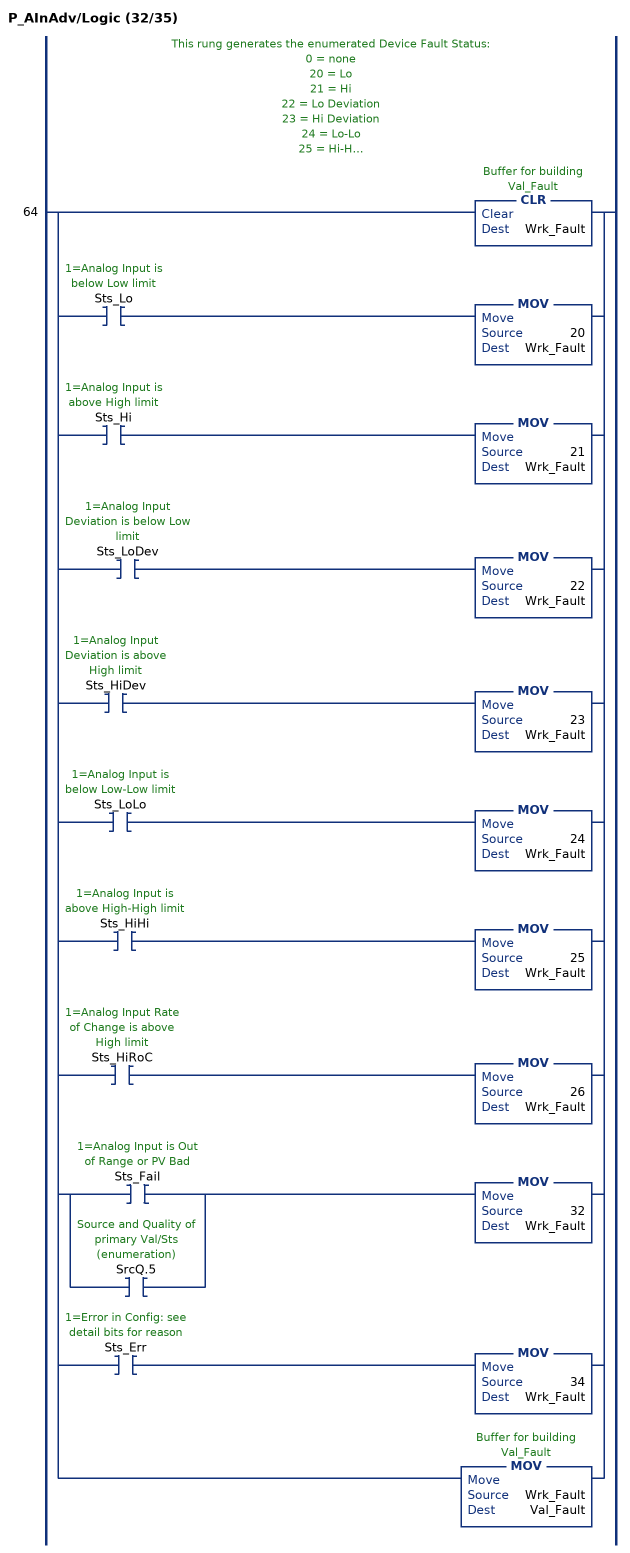
   // This rung generates the enumerated Device Fault Status:
   // 0 = none
   // 20 = Lo
   // 21 = Hi
   // 22 = Lo Deviation
   // 23 = Hi Deviation
   // 24 = Lo-Lo
   // 25 = Hi-Hi
   // 26 = Hi Rate of Change
   // 32 = Failed (I/O fault or out of range)
   // 34 = Config Error
   64: [CLR(Wrk_Fault) ,XIC(Sts_Lo) MOV(20,Wrk_Fault) ,XIC(Sts_Hi) MOV(21,Wrk_Fault) ,XIC(Sts_LoDev) MOV(22,Wrk_Fault) ,XIC(Sts_HiDev) MOV(23,Wrk_Fault) ,XIC(Sts_LoLo) MOV(24,Wrk_Fault) ,XIC(Sts_HiHi) MOV(25,Wrk_Fault) ,XIC(Sts_HiRoC) MOV(26,Wrk_Fault) ,[XIC(Sts_Fail) ,XIC(SrcQ.5) ] MOV(32,Wrk_Fault) ,XIC(Sts_Err) MOV(34,Wrk_Fault) ,MOV(Wrk_Fault,Val_Fault) ];
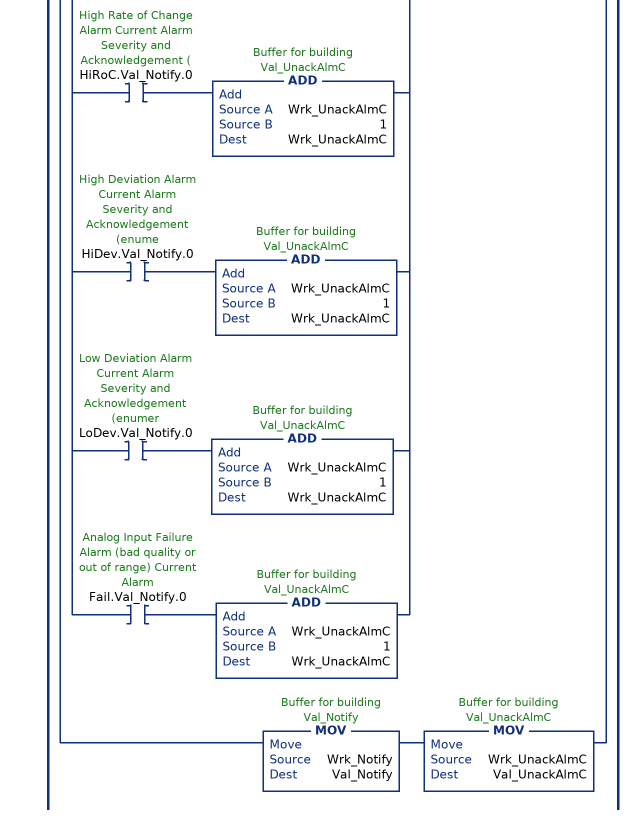
   // ============================================================
   // NOTIFICATION VALUE
   // ============================================================
   // Indicate the current alarm notification level as the max of any of the alarms,
   // and set the low-order bit for reset or ack required:
   // 0 = Not in alarm, acknowledged
   // 1 = Not in alarm, unacknowledged or reset required
   // 2 = Low severity alarm, acknowledged
   // 3 = Low severity alarm, unacknowledged
   // 4 = Medium severity alarm, acknowledged
   // 5 = Medium severity alarm, unacknowledged
   // 6 = High severity alarm, acknowledged
   // 7 = High severity alarm, unacknowledged
   // 8 = Urgent severity alarm, acknowledged
   // 9 = Urgent severity alarm, unacknowledged
   // #####  V4.00.00  2018-06-25:  Added Val_NotifyAll and Val_UnackAlmC to roll up alarm  #####
   // #####  priority / ack status and unack. alarm count including attached Channel object.  #####
   65: [CLR(Wrk_Notify) CLR(Wrk_UnackAlmC) OTU(Wrk_Notify.0) ,GRT(HiHi.Val_Notify,Wrk_Notify) MOV(HiHi.Val_Notify,Wrk_Notify) ,GRT(Hi.Val_Notify,Wrk_Notify) MOV(Hi.Val_Notify,Wrk_Notify) ,GRT(Lo.Val_Notify,Wrk_Notify) MOV(Lo.Val_Notify,Wrk_Notify) ,GRT(LoLo.Val_Notify,Wrk_Notify) MOV(LoLo.Val_Notify,Wrk_Notify) ,GRT(HiRoC.Val_Notify,Wrk_Notify) MOV(HiRoC.Val_Notify,Wrk_Notify) ,GRT(HiDev.Val_Notify,Wrk_Notify) MOV(HiDev.Val_Notify,Wrk_Notify) ,GRT(LoDev.Val_Notify,Wrk_Notify) MOV(LoDev.Val_Notify,Wrk_Notify) ,GRT(Fail.Val_Notify,Wrk_Notify) MOV(Fail.Val_Notify,Wrk_Notify) ,[XIC(HiHi.Val_Notify.0) ADD(Wrk_UnackAlmC,1,Wrk_UnackAlmC) ,XIC(Hi.Val_Notify.0) ADD(Wrk_UnackAlmC,1,Wrk_UnackAlmC) ,XIC(Lo.Val_Notify.0) ADD(Wrk_UnackAlmC,1,Wrk_UnackAlmC) ,XIC(LoLo.Val_Notify.0) ADD(Wrk_UnackAlmC,1,Wrk_UnackAlmC) ,XIC(HiRoC.Val_Notify.0) ADD(Wrk_UnackAlmC,1,Wrk_UnackAlmC) ,XIC(HiDev.Val_Notify.0) ADD(Wrk_UnackAlmC,1,Wrk_UnackAlmC) ,XIC(LoDev.Val_Notify.0) ADD(Wrk_UnackAlmC,1,Wrk_UnackAlmC) ,XIC(Fail.Val_Notify.0) ADD(Wrk_UnackAlmC,1,Wrk_UnackAlmC) ] OTL(Wrk_Notify.0) ,MOV(Wrk_Notify,Val_Notify) MOV(Wrk_UnackAlmC,Val_UnackAlmC) ];
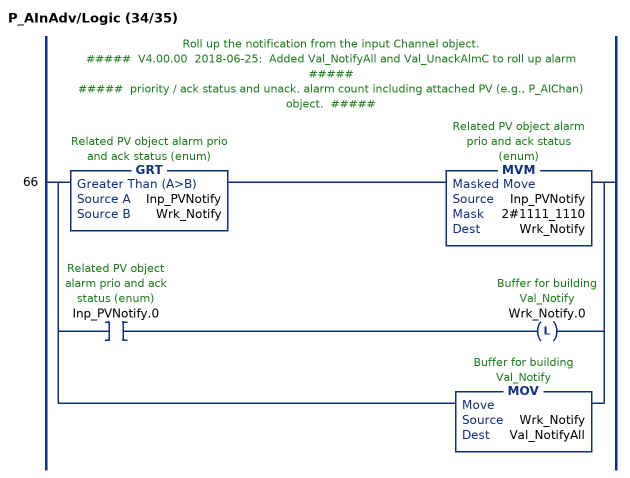
   // Roll up the notification from the input Channel object.
   // #####  V4.00.00  2018-06-25:  Added Val_NotifyAll and Val_UnackAlmC to roll up alarm  #####
   // #####  priority / ack status and unack. alarm count including attached PV (e.g., P_AIChan) object.  #####
   66: [GRT(Inp_PVNotify,Wrk_Notify) MVM(Inp_PVNotify,2#1111_1110,Wrk_Notify) ,XIC(Inp_PVNotify.0) OTL(Wrk_Notify.0) ,MOV(Wrk_Notify,Val_NotifyAll) ];
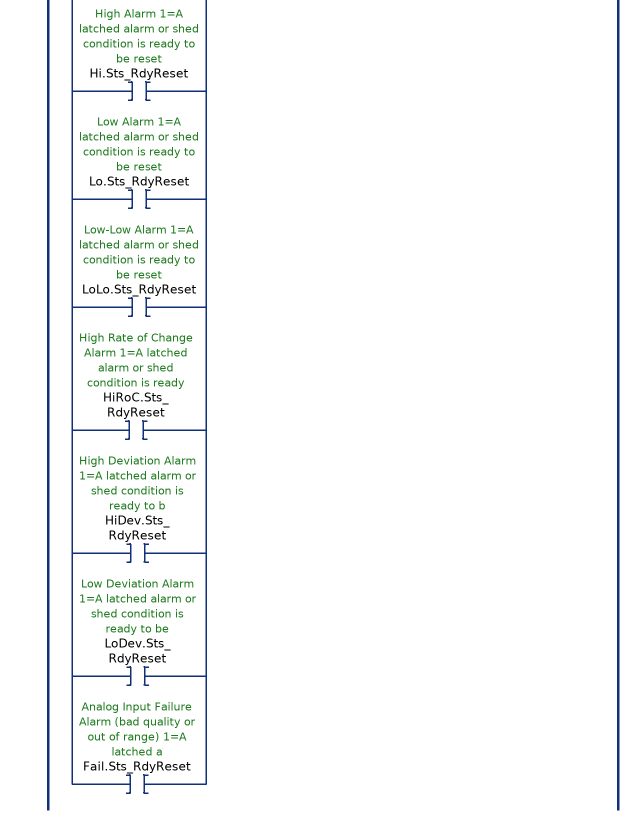
   // This rung identifies:
   // * if any alarm reset or other reset is required; and
   // * if any reset or acknowledge from the operator is required.
   // #####  V4.00.00  2018-06-25:  Aligned ready bit naming with command bit names.  #####
   // #####  All OCmds/MCmds and ORdys/MRdys are now Local Tags.  #####
   // #####  Added Sts_RdyAck and Sts_ResetReqd for use by external objects.  #####
   67: [[XIC(HiHi.Sts_RdyAck) ,XIC(Hi.Sts_RdyAck) ,XIC(Lo.Sts_RdyAck) ,XIC(LoLo.Sts_RdyAck) ,XIC(HiRoC.Sts_RdyAck) ,XIC(HiDev.Sts_RdyAck) ,XIC(LoDev.Sts_RdyAck) ,XIC(Fail.Sts_RdyAck) ] OTE(Sts_RdyAck) ,[XIC(HiHi.Sts_RdyReset) ,XIC(Hi.Sts_RdyReset) ,XIC(Lo.Sts_RdyReset) ,XIC(LoLo.Sts_RdyReset) ,XIC(HiRoC.Sts_RdyReset) ,XIC(HiDev.Sts_RdyReset) ,XIC(LoDev.Sts_RdyReset) ,XIC(Fail.Sts_RdyReset) ] OTE(ORdy_Reset) ]OTE(ORdy_ResetAckAll);
END_ROUTINE
